FUNCTION_BLOCK TestMotion
VAR_IN_OUT
	axisXP  : AXIS_REF; //Axis 1;
	axisXM : AXIS_REF; //Axis 2;
	nextInstruct, abortRequest, resetRequest, startRequest, stopRequest: BOOL;
	homeRequest : BYTE;
		
	//statemachine
	state : INT;
	
END_VAR
VAR_INPUT

	speed : LREAL;	

END_VAR
VAR_OUTPUT
END_VAR
VAR
	
	//power 
	mcPowerXP : MC_Power;
	mcPowerXM : MC_Power;
	mcResetXP : MC_Reset;
	mcResetXM : MC_Reset;
	
	//motion
	mcMoveAbsXP : MC_MoveAbsolute;
	mcMoveAbsXM : MC_MoveAbsolute;
	mcHomeXP 	: MC_Home;
	mcHomeXM 	: MC_Home;
	mcHalt		: MC_Halt;
	
	//Direction
	directionXP : BOOL;
	
	//position
	mcSetPosXP : MC_SetPosition;
	mcSetPosXM : MC_SetPosition;
	
	//error var
	errorIDXP : UDINT;
	errorIDXM : UDINT;
	
	//calibration var
	hallSigCalXP_rtrig	: ARRAY [GVL.HALL_LL_XP_C .. GVL.HALL_UL_XP_C] OF  R_TRIG;
	hallSigCalXP_ftrig 	: ARRAY [GVL.HALL_LL_XP_C .. GVL.HALL_UL_XP_C] OF  F_TRIG;
	hallSigCalXM_rtrig	: ARRAY [GVL.HALL_LL_XM_C .. GVL.HALL_UL_XM_C] OF  R_TRIG;
	hallSigCalXM_ftrig 	: ARRAY [GVL.HALL_LL_XM_C .. GVL.HALL_UL_XM_C] OF  F_TRIG;
	
	//r_Trig var
	hallSigAct_rtrig	: R_TRIG;
	hallSigAct_ftrig 	: F_TRIG;
	
	//counter
	iReset 	: INT :=0;
	jReset	: INT :=0;
	iCal	: INT :=0;
	jCal	: INT :=0;
	iPos	: INT :=0;
	jPos	: INT :=0;
	tripCountXP : ARRAY[GVL.HALL_LL_XP_C .. GVL.HALL_UL_XP_C] OF INT; //12 hall switch per blade
	tripCountXM : ARRAY[0..12] OF INT; //12 hall switch per blade

	//Test Var
	testVar : INT :=0;
	
END_VAR
VAR CONSTANT
	BRAKES_OFF_C	: BYTE	:= 3;
	BRAKES_ON_C		: BYTE	:= 0;
	HOME_VEL_C		: LREAL	:= 30;
	CALIBRATE_VEL_C	: LREAL	:= 60;
	POSITION_VEL_C	: LREAL := 300;
	POS_START_C		: LREAL := 0;
	POS_END_C		: LREAL := 750;
	HOMEOFFSET_XP_C	: LREAL	:= (POS_START_C+35);
	HOMEOFFSET_XM_C	: LREAL	:= (POS_END_C-85);
	
	SIZE_HALL_SW_C 	: LREAL := SIZEOF(GVL.hallPosCalXP);
END_VAR

axisXP.ReadStatus();
axisXM.ReadStatus();


//reset input
IF abortRequest THEN
	abortRequest := FALSE;
	state := -1; //stop state
END_IF
IF resetRequest THEN
	resetRequest := FALSE;
	state := 0;
END_IF

//Homing selection block
IF homeRequest=1 THEN
	state := 200;
ELSIF homeRequest=2 THEN
	state := 300;
ELSIF homeRequest=3 THEN
	state := 400;
END_IF
homeRequest := 0;

//if brakes are not disengaged, disable axis movement
IF GVL.brakeRelays <> 3 THEN
	McPowerXP(Axis := axisXP, Enable := TRUE, Enable_Positive := FALSE, Enable_Negative := FALSE);
	McPowerXM(Axis := axisXM, Enable := TRUE, Enable_Positive := FALSE, Enable_Negative := FALSE);
ELSE
	McPowerXP(Axis := axisXP, Enable := TRUE, Enable_Positive := TRUE, Enable_Negative := TRUE);
	McPowerXM(Axis := axisXM, Enable := TRUE, Enable_Positive := TRUE, Enable_Negative := TRUE); 
END_IF

//if any of the axis is not homed, disable other movement state until homed
IF state>420 THEN
	IF NOT axisXP.Status.Homed OR NOT axisXM.Status.Homed THEN
		abortRequest:=TRUE;
	END_IF
END_IF


CASE state OF
	-1: //Abort state. Disable movement
		McPowerXP(Axis := axisXP, Enable := TRUE, Enable_Positive := FALSE, Enable_Negative := FALSE);
		McPowerXM(Axis := axisXM, Enable := TRUE, Enable_Positive := FALSE, Enable_Negative := FALSE);
		mcHomeXP(Axis := axisXP, Execute := FALSE);
		mcHomeXM(Axis := axisXP, Execute := FALSE);
		nextInstruct := FALSE;
		GVL.brakeRelays := BRAKES_ON_C;
		GVL.fbWaitTimer(IN:=FALSE);
		
	0: //reset state
		nextInstruct := FALSE;
		mcResetXP(Axis := axisXP, Execute := TRUE, ErrorID => errorIDXP);
		mcResetXM(Axis := axisXM, Execute := TRUE, ErrorID => errorIDXM);
		IF mcResetXP.Error OR mcResetXM.Error THEN
			McPowerXP(Axis := axisXP, Enable := TRUE, Enable_Positive := FALSE, Enable_Negative := FALSE);
			McPowerXM(Axis := axisXM, Enable := TRUE, Enable_Positive := FALSE, Enable_Negative := FALSE);
			GVL.brakeRelays := BRAKES_ON_C;
			state 			:= 100; //go to stop state
		ELSIF mcResetXP.Done AND mcResetXM.Done THEN
			McPowerXP(Axis := axisXP, Enable := TRUE, Enable_Positive := TRUE, Enable_Negative := TRUE);
			McPowerXM(Axis := axisXM, Enable := TRUE, Enable_Positive := TRUE, Enable_Negative := TRUE);
			mcResetXP(Axis := axisXP, Execute := FALSE);
			mcResetXM(Axis := axisXM, Execute := FALSE);
			GVL.brakeRelays	:= BRAKES_OFF_C;
			state 			:= 100; //go to stop state
		END_IF

		
	100: //stop state
		mcMoveAbsXP(Axis := axisXP, Execute := FALSE);
		mcMoveAbsXM(Axis := axisXM, Execute := FALSE);
		mcHomeXP(Axis := axisXP, Execute := FALSE);
		mcHomeXM(Axis := axisXP, Execute := FALSE);
		GVL.fbWaitTimer(IN:=FALSE);

	
	
	400: //Homing start for both blades
		mcHomeXP(Axis := axisXP, Position := HOMEOFFSET_XP_C, bCalibrationCam := GVL.limitHomeXp, Execute := TRUE);
		mcHomeXM(Axis := axisXM, Position := HOMEOFFSET_XM_C, bCalibrationCam := GVL.limitHomeXm, Execute := TRUE);
		IF mcHomeXP.Done AND mcHomeXM.Done THEN
			state := 410;
		END_IF
		
	410: //Homing running for both blades
		IF NOT mcHomeXP.Error AND NOT mcHomeXM.Error THEN
			mcHomeXP(Axis := axisXP, Execute := FALSE);
			mcMoveAbsXP(Axis:=axisXP, Velocity:=HOME_VEL_C, Position:=POS_START_C, Execute:= TRUE,);
			mcHomeXM(Axis := axisXM, Execute := FALSE);
			mcMoveAbsXM(Axis:=axisXM, Velocity:=HOME_VEL_C, Position:=POS_END_C, Execute:= TRUE);
			IF mcMoveAbsXP.Done AND mcMoveAbsXM.Done THEN
				mcMoveAbsXP(Axis:=axisXP, Execute:= FALSE);
				mcMoveAbsXM(Axis:=axisXM, Execute:= FALSE);
				state := 100; 
			END_IF
		ELSE
			state :=100; //stop state. Should go to error state
		END_IF

	420: //Homing routine complete for AxisXM
		mcSetPosXP(Axis:=axisXP, Execute:=FALSE);
		mcSetPosXM(Axis:=axisXM, Execute:=FALSE);
		IF  mcSetPosXP.Done AND mcSetPosXM.Done THEN
			state := 100;
		END_IF	

//States higher than 420 requires HOMING ROUTINE to be run first.


//Basic Motions ---------------------------------------------------------------
	1000: //Open shutter
		mcMoveAbsXP(Axis:=axisXP, Position:= POS_START_C, Velocity:=speed, Execute:=TRUE);
		mcMoveAbsXM(Axis:=axisXM, Position:= POS_END_C, Velocity:=speed, Execute:=TRUE);
		IF mcMoveAbsXP.Done AND mcMoveAbsXM.Done THEN
			state:=100;
		END_IF
		
		
	1100: //Close shutter towards X+ side. AxisXP retracts to its HOME position
		mcMoveAbsXP(Axis:=axisXP, Position:= POS_START_C, Velocity:=speed, Execute:=TRUE);
		IF mcMoveAbsXP.Done THEN
			mcMoveAbsXP(Axis:=axisXP, Execute:=FALSE);
			state:=1110;
		END_IF
		
	1110: //Close shutter towards X+ side. AxisXM extends to its DEPLOYED position 
		mcMoveAbsXM(Axis:=axisXM, Position:= POS_START_C, Velocity:=speed, Execute:=TRUE);
		IF mcMoveAbsXM.Done THEN
			mcMoveAbsXM(Axis:=axisXM, Execute:=FALSE);
			state:=100;	
		END_IF
		
	1200: //Close shutter towards X- side. AxisXM retracts to its HOME position (~750 mm)
		mcMoveAbsXM(Axis:=axisXM, Position:= POS_END_C, Velocity:=speed, Execute:=TRUE);
		IF mcMoveAbsXM.Done THEN
			mcMoveAbsXM(Axis:=axisXM, Execute:=FALSE);
			state:=1210;
		END_IF
		
	1210: //Close shutter towards X- side. AxisXP extends to its DEPLOYED position
		mcMoveAbsXP(Axis:=axisXP, Position:= POS_END_C, Velocity:=speed, Execute:=TRUE);
		IF mcMoveAbsXP.Done THEN
			mcMoveAbsXP(Axis:=axisXP, Execute:=FALSE);
			state:=100;
		END_IF


//Motion for visit----------------------------------------------------------------------------
		
	2000: //Normal Visit. Put both blades in position at 0 mm - Shutter closed
		mcMoveAbsXP(Axis:=axisXP, Position:=POS_START_C, Velocity:=POSITION_VEL_C, Execute:=TRUE);
		IF mcMoveAbsXP.Done THEN
			mcMoveAbsXP(Axis:=axisXP, Execute:=FALSE);
			mcMoveAbsXM(Axis:=axisXM, Position:=POS_START_C, Velocity:=POSITION_VEL_C, Execute:=TRUE);
			IF  mcMoveAbsXM.Done THEN
				mcMoveAbsXM(Axis:=axisXM, Execute:=FALSE);
				state:=2010;
			END_IF	
		END_IF
	
	2010: //Normal Visit. Blade in position. Wait for input to continue.
		IF nextInstruct THEN
			nextInstruct:=FALSE;
			state:=2100;
		END_IF
		
	2100: //Normal Visit. Visit 1 sequence - axisXM travels to end of X- side after set time elapsed - Shutter open
		GVL.fbWaitTimer(IN:=TRUE, PT:=GVL.expoTime,);
		mcMoveAbsXM(Axis:=axisXM, Position:=POS_END_C, Velocity:=speed, Execute:=TRUE);
		IF mcMoveAbsXM.Done AND GVL.fbWaitTimer.Q THEN
			GVL.fbWaitTimer(IN:=FALSE);
			mcMoveAbsXM(Axis:=axisXM, Execute:=FALSE);
			state:=2110;
		END_IF

	2110: //Normal Visit. Visit 1 sequence - axisXP travels to end of X- side - Shutter close
		mcMoveAbsXP(Axis:=axisXP, Position:=POS_END_C, Velocity:=speed, Execute:=TRUE);
		IF mcMoveAbsXP.Done THEN
			mcMoveAbsXP(Axis:=axisXP, Execute:=FALSE);
			state:=2120;
		END_IF
		
	2120: //Normal Visit. Pause at the end of first visit. Wait for input to continue
		GVL.fbWaitTimer(IN:=TRUE, PT:=T#2S);
		IF nextInstruct OR GVL.fbWaitTimer.Q THEN
			GVL.fbWaitTimer(IN:=FALSE);
			nextInstruct:=FALSE;
			state:=2200;
		END_IF
	
	2200: //Normal Visit. Visit 2 sequence - axisXP travels to X+ side - Shutter open
		GVL.fbWaitTimer(IN:=TRUE, PT:=GVL.expoTime,);
		mcMoveAbsXP(Axis:=axisXP, Position:=POS_START_C, Velocity:=speed, Execute:=TRUE);
		IF mcMoveAbsXP.Done AND GVL.fbWaitTimer.Q THEN
			GVL.fbWaitTimer(IN:=FALSE);
			mcMoveAbsXP(Axis:=axisXP, Execute:=FALSE);
			state:=2210;
		END_IF
		
	2210: //Normal Visit. Visit 2 sequence - axisXM travels to X+ side - Shutter close
		mcMoveAbsXM(Axis:=axisXM, Position:=POS_START_C, Velocity:=speed, Execute:=TRUE);
		IF mcMoveAbsXM.Done THEN
			mcMoveAbsXM(Axis:=axisXM, Execute:=FALSE);
			state:=100;
		END_IF
		
//Cycler -- for use in testing shutter cycle
		
	3100: //Cycler sequence - axisXM travels to end of X- side after set time elapsed - Shutter open
		GVL.fbWaitTimer(IN:=TRUE, PT:=GVL.expoTime,);
		mcMoveAbsXM(Axis:=axisXM, Position:=POS_END_C, Velocity:=speed, Execute:=TRUE);
		IF mcMoveAbsXM.Done AND GVL.fbWaitTimer.Q THEN
			GVL.fbWaitTimer(IN:=FALSE);
			mcMoveAbsXM(Axis:=axisXM, Execute:=FALSE);
			state:=3110;
			IF stopRequest THEN
				stopRequest:=FALSE;
				state:=100;
			END_IF
		END_IF


	3110: //Cycler sequence - axisXP travels to end of X- side - Shutter close
		mcMoveAbsXP(Axis:=axisXP, Position:=POS_END_C, Velocity:=speed, Execute:=TRUE);
		IF mcMoveAbsXP.Done THEN
			mcMoveAbsXP(Axis:=axisXP, Execute:=FALSE);
			state:=3120;
			IF stopRequest THEN
				stopRequest:=FALSE;
				state:=100;
			END_IF
		END_IF
		
		
	3120: //Pause at the end of travel. Wait for input or timer to continue
		GVL.fbWaitTimer(IN:=TRUE, PT:=T#1S);
		IF nextInstruct OR GVL.fbWaitTimer.Q THEN
			GVL.fbWaitTimer(IN:=FALSE);
			nextInstruct:=FALSE;
			state:=3200;
			IF stopRequest THEN
				stopRequest:=FALSE;
				state:=100;
			END_IF
		END_IF
	
	3200: //axisXP travels to X+ side - Shutter open
		GVL.fbWaitTimer(IN:=TRUE, PT:=GVL.expoTime,);
		mcMoveAbsXP(Axis:=axisXP, Position:=POS_START_C, Velocity:=speed, Execute:=TRUE);
		IF mcMoveAbsXP.Done AND GVL.fbWaitTimer.Q THEN
			GVL.fbWaitTimer(IN:=FALSE);
			mcMoveAbsXP(Axis:=axisXP, Execute:=FALSE);
			state:=3210;
			IF stopRequest THEN
				stopRequest:=FALSE;
				state:=100;
			END_IF
		END_IF
		
	3210: //axisXM travels to X+ side - Shutter close
		mcMoveAbsXM(Axis:=axisXM, Position:=POS_START_C, Velocity:=speed, Execute:=TRUE);
		IF mcMoveAbsXM.Done THEN
			mcMoveAbsXM(Axis:=axisXM, Execute:=FALSE);
			state:=3220;
			IF stopRequest THEN
				stopRequest:=FALSE;
				state:=100;
			END_IF
		END_IF
		
	3220: //Pause at the end of travel. Wait for input or timer to continue
		GVL.fbWaitTimer(IN:=TRUE, PT:=T#1S);
		IF nextInstruct OR GVL.fbWaitTimer.Q THEN
			GVL.fbWaitTimer(IN:=FALSE);
			nextInstruct:=FALSE;
			state:=3100;
			IF stopRequest THEN
				stopRequest:=FALSE;
				state:=100;
			END_IF
		END_IF
		

//Calibration -----------------------------------------------------------------------------
	9000: //Clear previous Calibration value
		FOR iReset:=GVL.HALL_LL_XP_C TO GVL.HALL_UL_XP_C BY 1 DO
			FOR jReset:=0 TO GVL.HALL_TRIP_C BY 1 DO
				GVL.hallPosCalXP[0,iReset, jReset]:=0;
				GVL.hallPosCalXP[1,iReset, jReset]:=0;
			END_FOR
		END_FOR
		FOR iPos:=GVL.HALL_LL_XP_C TO GVL.HALL_UL_XP_C BY 1 DO
				tripCountXP[iPos] := 0;		
		END_FOR
		state:=9010;
		
	9010: //Put Shutter in Open Position
		mcMoveAbsXP(Axis:=axisXP, Position:= POS_START_C, Velocity:=POSITION_VEL_C, Execute:=TRUE);
		mcMoveAbsXM(Axis:=axisXM, Position:= POS_END_C, Velocity:=POSITION_VEL_C, Execute:=TRUE);
		IF mcMoveAbsXP.Done AND mcMoveAbsXM.Done THEN
			mcMoveAbsXP(Axis:=axisXP, Execute:=FALSE);
			state:=9020;
		END_IF
		//This section is required to get rid of false trigger when system starts up

		FOR iCal:=GVL.HALL_LL_XP_C TO GVL.HALL_UL_XP_C BY 1 DO
			hallSigCalXP_rtrig[iCal](CLK:=GVL.hallSwitch[iCal]);
			hallSigCalXP_ftrig[iCal](CLK:=GVL.hallSwitch[iCal]);
			IF hallSigCalXP_rtrig[iCal].Q OR hallSigCalXP_ftrig[iCal].Q THEN
				;
			END_IF
		END_FOR

	9020: //Calibrate AxisXP towards X- side.
		//record hall trips at rising and falling edge
		FOR iCal:=GVL.HALL_LL_XP_C TO GVL.HALL_UL_XP_C BY 1 DO
			hallSigCalXP_rtrig[iCal](CLK:=GVL.hallSwitch[iCal]);
			hallSigCalXP_ftrig[iCal](CLK:=GVL.hallSwitch[iCal]);
			IF hallSigCalXP_rtrig[iCal].Q OR hallSigCalXP_ftrig[iCal].Q THEN
				
				GVL.hallPosCalXP[0, iCal, tripCountXP[iCal]] := axisXP.NcToPlc.ActPos;
				tripCountXP[iCal] := tripCountXP[iCal] + 1;
				//IF tripCountXP[iCal]>15 THEN
					//tripCountXP[iCal]:=0;
				//END_IF
				
			END_IF
		END_FOR
	
		//start moving axisXP towards x- side
		mcMoveAbsXP(Axis:=axisXP, Position:=POS_END_C, Velocity:=CALIBRATE_VEL_C, Execute:=TRUE);
		IF mcMoveAbsXP.Done THEN
			mcMoveAbsXP(Axis:=axisXP, Execute:=FALSE);
			state:= 9030;
		END_IF
	
		9030: //Calibrate AxisXP towards X+ side.
		//record hall trips at rising and falling edge
		FOR iCal:=GVL.HALL_LL_XP_C TO GVL.HALL_UL_XP_C BY 1 DO
			hallSigCalXP_rtrig[iCal](CLK:=GVL.hallSwitch[iCal]);
			hallSigCalXP_ftrig[iCal](CLK:=GVL.hallSwitch[iCal]);
			IF hallSigCalXP_rtrig[iCal].Q OR hallSigCalXP_ftrig[iCal].Q THEN
				
				GVL.hallPosCalXP[1, iCal, tripCountXP[iCal]] := axisXP.NcToPlc.ActPos;
				tripCountXP[iCal] := tripCountXP[iCal] - 1;
				//IF tripCountXP[iCal]>15 THEN
					//tripCountXP[iCal]:=0;
				//END_IF
				
			END_IF
		END_FOR
	
		//start moving axisXP towards x+ side
		mcMoveAbsXP(Axis:=axisXP, Position:=POS_START_C, Velocity:=CALIBRATE_VEL_C, Execute:=TRUE);
		IF mcMoveAbsXP.Done THEN
			mcMoveAbsXP(Axis:=axisXP, Execute:=FALSE);
			state:= 9040;
		END_IF
		
		
	
	9040: //Put shutter in open position after calibration
		mcMoveAbsXP(Axis:=axisXP, Position:= POS_START_C, Velocity:=POSITION_VEL_C, Execute:=TRUE);
		mcMoveAbsXM(Axis:=axisXM, Position:= POS_END_C, Velocity:=POSITION_VEL_C, Execute:=TRUE);
		IF mcMoveAbsXP.Done AND mcMoveAbsXM.Done THEN
			mcMoveAbsXP(Axis:=axisXP, Execute:=FALSE);
			state:=100;
		END_IF
END_CASE


//Actual Position Calc
FOR iPos:=GVL.HALL_LL_XP_C TO GVL.HALL_UL_XP_C BY 1 DO
	hallSigCalXP_rtrig[iPos](CLK:=GVL.hallSwitch[iPos]);
	hallSigCalXP_ftrig[iPos](CLK:=GVL.hallSwitch[iPos]);
	IF hallSigCalXP_rtrig[iPos].Q OR hallSigCalXP_ftrig[iPos].Q THEN
		IF axisXP.status.PositiveDirection THEN
			GVL.hallPosActXP := GVL.hallPosCalXP[0, iPos, tripCountXP[iPos]];
			tripCountXP[iPos] := tripCountXP[iPos] + 1;	
		END_IF
		IF axisXP.status.NegativeDirection THEN
			GVL.hallPosActXP := GVL.hallPosCalXP[1, iPos, tripCountXP[iPos]];
			tripCountXP[iPos] := tripCountXP[iPos] - 1;	
		END_IF
	END_IF
END_FOR

(* //Reset trip counter
IF axisXP.Status.InPositionArea AND state<9000 THEN
	FOR iPos:=GVL.HALL_LL_XP_C TO GVL.HALL_UL_XP_C BY 1 DO
		tripCountXP[iPos] := 0;		
	END_FOR
END_IF 
*)

END_FUNCTION_BLOCK

(* stored: Version 1.1.0.1, ProductVersion 3.1.4020.12
   POU TestMotion: Id {f5ec753e-2f53-4143-ab85-291d0817da2d}, SpecialFunc None *)
